// TIA Portal V19 export
TYPE "ValveMachine_DataIn"
// stored: Access Published
   STRUCT
      PB : "ValveMachine_PB";   // Pulsanti manuali
      Rest_Ls : Array[1..8] of Bool;   // Finecorsa REST
      Work_Ls : Array[1..8] of Bool;   // Finecorsa WORK
   END_STRUCT;
END_TYPE
